# B&R Automation Studio project pp70debox_Vision
Automation Studio 4.6.3.55 SP

## Configuration Config1

CPU 4PPC70.0702-20B, AutomationRuntime B4.62, Build 4.1.2, Vc V4.62.0

### Task classes (Cpu.sw)
```
Cyclic#4:
  Camera <- Camera.prg
  Program <- Program.prg
VcDataObjects: VisuPP <- VisuPP70sync.dob
```

### Hardware
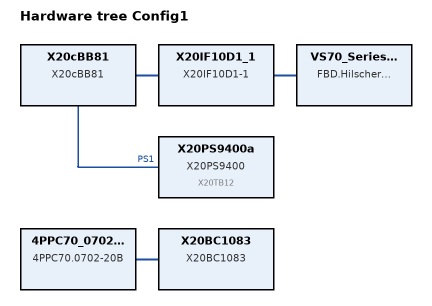
```
4PPC70_0702_20B : 4PPC70.0702-20B v1.4.0.0
  Connector IF2:
    ActivateDevice = 1
    Mode = Manual
    InternetAddress = 10.16.7.36
    SubnetMask = 255.255.0.0
    DeviceParam = /EDDN=gei
  ConfigurationID = pp500_Config1
  ActivateOpcUa = 1
  OpcUaInformationModels_PV_Version = 1
  VcObjectName = VisuPP
  KeyMappingFile = VC\4PPC70_0702_20B.dis
VS70_Series_V11_1 : FBD.Hilscher.EIGenEDSAdapterDTM.VS70 Series V11.1 v11.1 (OrderNumber=VS70 Series V11.1, VendorAddress=10.16.7.19)  [EIP1 -> X20IF10D1_1.IF1]
  DtmId = 6f05449d-88db-4399-ac96-feab6093c4e0
  ChannelBlocks_4b4b5f3d-aef6-4330-98f3-b7c28e4e6291  // Module 0
  IO_InputImage_4b4b5f3d-aef6-4330-98f3-b7c28e4e6291  // 496 Byte(s)
  Channel_1_IO_InputImage_4b4b5f3d-aef6-4330-98f3-b7c28e4e6291
  Name_Channel_1_IO_InputImage_4b4b5f3d-aef6-4330-98f3-b7c28e4e6291 = Angle  // Angle du cercle
  Type_Channel_1_IO_InputImage_4b4b5f3d-aef6-4330-98f3-b7c28e4e6291 = INT
  Channel_2_IO_InputImage_4b4b5f3d-aef6-4330-98f3-b7c28e4e6291
  Name_Channel_2_IO_InputImage_4b4b5f3d-aef6-4330-98f3-b7c28e4e6291 = X
  Type_Channel_2_IO_InputImage_4b4b5f3d-aef6-4330-98f3-b7c28e4e6291 = INT
  Channel_3_IO_InputImage_4b4b5f3d-aef6-4330-98f3-b7c28e4e6291
  Name_Channel_3_IO_InputImage_4b4b5f3d-aef6-4330-98f3-b7c28e4e6291 = Y  // Coordonnée Y
  Type_Channel_3_IO_InputImage_4b4b5f3d-aef6-4330-98f3-b7c28e4e6291 = INT
  Channel_4_IO_InputImage_4b4b5f3d-aef6-4330-98f3-b7c28e4e6291
  Name_Channel_4_IO_InputImage_4b4b5f3d-aef6-4330-98f3-b7c28e4e6291 = Diametre  // Diamètre du cercle
  Type_Channel_4_IO_InputImage_4b4b5f3d-aef6-4330-98f3-b7c28e4e6291 = INT
  IO_OutputImage_4b4b5f3d-aef6-4330-98f3-b7c28e4e6291  // 496 Byte(s)
X20BC1083 : X20BC1083 v2.7.0.0  [PLK2 -> 4PPC70_0702_20B.IF1 (NodeNumber=2) [Cable Type=PowerlinkCable, Length=10, Version=1.0.0.2]; SL -> X20cBB81.SL1]
  Supervision = off
X20IF10D1_1 : X20IF10D1-1 v1.3.1.0  [SS -> X20cBB81.SS1]
  Connector IF1:
    DtmRef = FBDIF.Hilscher.ENIPScannerDTM.NETX 100 RE/EIM
    DtmId = ff88a3d9-25be-4a21-a04e-17ce51bc7424
  ConfigFile = X20IF10D1_1.dtm
  ConfigModule = asnxdb1
X20PS9400a : X20PS9400 v1.0.2.4  [SS1 -> X20TB12a.SS; PS -> X20cBB81.PS1]
  Supervision = off
X20TB12a : X20TB12 v1.0.0.0
X20cBB81 : X20cBB81 v1.0.2.0
```

### IoMap.iom - 4PPC70_0702_20B/IoMap.iom
```iecst
VAR_CONFIG
	::Camera:Y AT %IW."VS70_Series_V11_1".Y;
	::Camera:X AT %IW."VS70_Series_V11_1".X;
	::Camera:Angle AT %IW."VS70_Series_V11_1".Angle;
	::Camera:Diametre AT %IW."VS70_Series_V11_1".Diametre;
	::Camera:Angle AT %ID."VS70_Series_V11_1".Angle;
	::Camera:Diametre AT %ID."VS70_Series_V11_1".Diametre;
	::Camera:Y AT %ID."VS70_Series_V11_1".Y;
	::Camera:X AT %ID."VS70_Series_V11_1".X;
END_VAR
```

## Logical view

### Program Logical/Camera (IEC)

#### Variables.var
```iecst
VAR
	Diametre : INT;
	tmpVar : REAL;
	X : INT;
	Y : INT;
	Z : INT;
	Angle : INT;
END_VAR
```

- Visualisation Logical/VisuPP70sync (not shown)

### Program Logical/Program (IEC)

#### Main.ab - Init, cyclic, exit code
```automation-basic
PROGRAM _INIT
	(* Insert code here *)

END_PROGRAM

PROGRAM _CYCLIC
	(* Insert code here *)

END_PROGRAM

PROGRAM _EXIT
	(* Insert code here *)

END_PROGRAM
```

#### Variables.var - Local variables
```iecst
VAR
	USINT_1_BR_COGNEX : USINT;
END_VAR
```

Listed in the project but not available here: Logical/Global.typ, Logical/Global.var, Logical/Libraries, Logical/Program/Types.typ
